// TIA Portal V17 export
// export: Created 2024-12-18T13:22:00.8190607Z, ExportSetting WithDefaults, DisplayName Totally Integrated Automation Portal, DisplayVersion V17 Update 6, DisplayName TIA Portal Openness, DisplayVersion V17 Update 6, DisplayName TIA Portal Version Control Interface, DisplayVersion V17, DisplayName SINAMICS Startdrive Advanced, DisplayVersion V17 SP1, DisplayName SINAMICS Startdrive G130, G150, S120, S150, SINAMICS MV, S210, DisplayVersion V17 SP1, DisplayName SINAMICS Startdrive G110M, G120, G120C, G120D, G120P, G115D, DisplayVersion V17 SP1, DisplayName STEP 7 Professional, DisplayVersion V17 Update 6, DisplayName SINUMERIK ONE STEP 7 Toolbox, DisplayVersion V17 Update 2, DisplayName SINUMERIK 840D sl STEP 7 Toolbox, DisplayVersion V17 Update 2, DisplayName STEP 7 Safety, DisplayVersion V17 Update 6, DisplayName WinCC Advanced / Unified PC, DisplayVersion V17 Update 6
FUNCTION "FC_LAD_Operations" : Void   // FC1, LAD
{ S7_Optimized_Access := 'TRUE' }
VERSION : 0.1
// stored: AutoNumber true, IsIECCheckEnabled false, SetENOAutomatically false, UDAEnableTagReadback false
   VAR_INPUT
      iSwitch1 : Bool;
      iSwitch2 : Bool;
   END_VAR
   VAR_OUTPUT
      qOutput : Bool;
   END_VAR
BEGIN

REGION Network 1
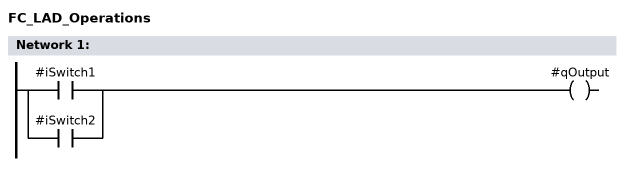
   RUNG wire#powerrail
      Contact( #iSwitch1 )
      wire#w1
      Coil( #qOutput )
   END_RUNG
   RUNG wire#powerrail
      Contact( #iSwitch2 )
   END_RUNG wire#w1
   // the same network as SCL:
   #qOutput := #iSwitch1 OR #iSwitch2;
END_REGION
END_FUNCTION
